SUBAPPLICATION logiBUS_AI_Calibrate_3P_Remote_IDA_OPC (* 3-Punkt-Kalibrierung (AR_CALIBRATE_3P_REF, unabhaengig gespeicherte Rohwerte X_MIN/X_MID/X_MAX + Referenzwerte MIN_REF/MID_REF/MAX_REF alle INI-persistiert) auf VT-Zahlenfelder (Rohwert + kalibrierter Wert, je eigene CNumberVariable) + Bargraph (kalibriert) + 3 VT-Tasten (C_MIN/C_MID/C_MAX) + OPC-UA (Rohwert DWORD + kalibrierter Wert REAL, generisch, ein Kanal). Wie logiBUS_AI_Calibrate_3P_IDA_OPC, aber der Rohwert kommt per Remote-Subscribe (AD_SUBSCRIBE_1) statt von einem lokalen logiBUS_AI_IDA - fuer Sensoren, deren physischer Analog-Eingang auf einer Station OHNE VT-Anschluss sitzt (z.B. Hangausgleich-Winkelsensor B14 auf APIXON STG3, waehrend Kalibrierung+VT auf der Station mit VT-Anschluss laufen). Der Rohwert wird dort per logiBUS_AI_Raw_Publish_OPC publiziert. *)
  (* Standard: 61499-2; Description: Copyright (c) 2026 Meisterschulen am Ostbahnhof This program and the accompanying materials are made available under the terms of the Eclipse Public License 2.0 which is available at https://www.eclipse.org/legal/epl-2.0/ SPDX-License-Identifier: EPL-2.0 *)
  (* Version 1.3, 2026-09-18, Franz Höpfinger, Meisterschulen am Ostbahnhof, AR_CALIBRATE_3P_REF.C_MIN/C_MID/C_MAX von AX-Sockets auf reine EventInputs umgestellt (Franz-Entscheidung, siehe AR_CALIBRATE_2P_REF) - AX_BOOL_TO_X_MIN/_MID/_MAX entfallen ersatzlos, die Merge-Ketten verbinden jetzt direkt per EventConnection mit CALIBRATE.C_MIN/C_MID/C_MAX. *)
  (* Version 1.4, 2026-09-18, Franz Höpfinger, Meisterschulen am Ostbahnhof, C_MIN/C_MAX-Merge-Ketten (2x E_MERGE_2 in Reihe) durch je einen E_MERGE_3 ersetzt, C_MID-Kette (3x E_MERGE_2) durch einen E_MERGE_4 - OR-Merge ist assoziativ, funktional identisch. Siehe logiBUS_AI_Calibrate_IDA_OPC v1.4. *)
  (* Version 1.2, 2026-09-16, Franz Höpfinger, Meisterschulen am Ostbahnhof, Fix (4diac-IDE-Validierungsfehler 'Cannot convert from AR2 to AR'): MID_REF_LIT.VALUEO/MAX_REF_LIT.VALUEO sind bidirektionale AR2-Plugs (Live-VT-Edit + Persistierung), kein einfacher AR-Wert wie CALIBRATE.Y - ein AR_SPLIT_2 direkt dazwischen ist falsch. MIDREF_OUT/MAXREF_OUT werden jetzt stattdessen von den neuen VALUE_OUT-Plugs auf MID_REF_LIT/MAX_REF_LIT gespeist (NumericValue_TO_AR2_OPC Version 1.1, plain-AR-Spiegel des Werts, unabhaengig vom bidirektionalen VALUEO). CAL_OUT (AR_SPLIT_3 auf CALIBRATE.Y, einfacher AR-Wert) war von diesem Fehler nicht betroffen und bleibt unveraendert. *)
  (* Version 1.1, 2026-09-16, Franz Höpfinger, Meisterschulen am Ostbahnhof, Neue optionale Ausgangs-Plugs CAL_OUT/MIDREF_OUT/MAXREF_OUT ergaenzt (AR_SPLIT_2 zu AR_SPLIT_3 fuer CAL, je 1 neuer AR_SPLIT_2 fuer MIDREF/MAXREF dazwischengesetzt) - damit externe Consumer (z.B. Fuellband_Oben_Erkennung/Befuellautomatik fuer den Fuellband-Kanal) den bereits kalibrierten Wert per Adapterverbindung lesen koennen statt selbst nochmal denselben OPC-UA-Knoten lokal zu abonnieren (FORTE: 'Cannot add another one'). Unverdrahtet lassen, wenn nicht gebraucht (z.B. Hangausgleich-Kanal). Siehe BERICHT_2026-09-16_STG3_I1_I3_I4_I6_STALE_REMOTE_SUBSCRIBE.md Abschnitt 16-17 Gruppe C. *)
  (* Version 1.0, 2026-09-11, Franz Höpfinger, Meisterschulen am Ostbahnhof, Remote-Rohwert-Variante von logiBUS_AI_Calibrate_3P_IDA_OPC - logiBUS_AI_IDA+AD_SPLIT_2+AD_PUBLISH_RAW durch AD_SUBSCRIBE_1 ersetzt, Rest der Kalibrier-/VT-Kette unveraendert. Fuer Hangausgleich-Winkelsensor B14 (STG3), Kalibrierung+VT auf STG1. *)
  (* Version 1.6, 2026-09-21, Franz Höpfinger, Meisterschulen am Ostbahnhof, Code-Review-Fund (PR #260): INI_X_MID/INI_X_MAX.DEFAULT_VALUE standen auf REAL#0.5/1.0 statt 0.0 - AR_CALIBRATE_3P_REF's xMidCal/xMaxCal-Kalibriert-Flags latchten dadurch bei JEDEM Boot sofort TRUE, obwohl MID/MAX nie kalibriert wurden. Defaults auf REAL#0.0 korrigiert. Betrifft Hangausgleich. *)
  (* Version 1.5, 2026-09-21, Franz Höpfinger, Meisterschulen am Ostbahnhof, AR_CALIBRATE_3P_REF hat jetzt ein INIT/QI/QO-Enable-Pattern (Bugfix MIN-vor-MID + xClipping) - CALIBRATE bekommt Parameter QI=TRUE, sonst bleibt die FB im START-Zustand haengen und REQ laeuft nie. *)
  PACKAGE MyLib::sys;
  IMPORT isobus::UT::Q::const::IDs::ID_NULL;
  IMPORT logiBUS::utils::conversion::phys::NumericObjectPool_S;
  IMPORT isobus::UT::io::Button::ButtonActivationCode::BT_PRESSED_LATCHED;
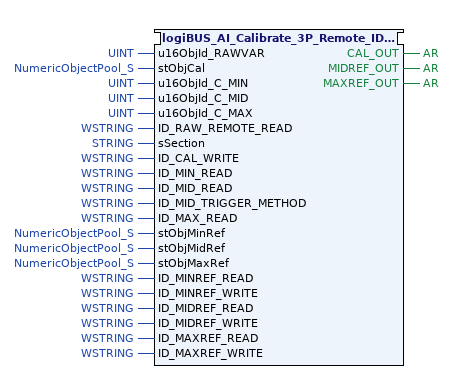
  VAR_INPUT
    u16ObjId_RAWVAR : UINT := ID_NULL; (* Object ID CNumberVariable (Rohwert 0-4095, unkalibriert, reine Diagnose-Anzeige) *)
    stObjCal : logiBUS::utils::conversion::phys::NumericObjectPool_S := (u16ObjId := ID_NULL, r32Scale := 1.0, i32Offset := 0, u8Decimals := 1); (* Object ID + Scale/Offset/Decimals CNumberVariable (kalibrierter Wert, eigene, unabhaengige CNumberVariable) *)
    u16ObjId_C_MIN : UINT := ID_NULL; (* Object ID Taste 'C_MIN' (Min-Position anfahren, dann druecken) *)
    u16ObjId_C_MID : UINT := ID_NULL; (* Object ID Taste 'C_MID' (Mittelstellung anfahren, dann druecken) *)
    u16ObjId_C_MAX : UINT := ID_NULL; (* Object ID Taste 'C_MAX' (Max-Position anfahren, dann druecken) *)
    ID_RAW_REMOTE_READ : WSTRING; (* Remote-Subscribe-Adresse des Rohwerts (DWORD 0-4095, ACTION=SUBSCRIBE) - Gegenstueck zu ID_RAW_WRITE auf der Sensor-Station (logiBUS_AI_Raw_Publish_OPC) *)
    sSection : STRING; (* INI-Sektionsname fuer X_MIN/X_MID/X_MAX/MIN_REF/MID_REF/MAX_REF-Persistenz - pro Kanal eindeutig, sonst kollidieren die Kanaele in settings.ini *)
    ID_CAL_WRITE : WSTRING; (* Kalibrierter-Wert-Ruckmelde-Adresse (REAL, ACTION=PUBLISH) *)
    ID_MIN_READ : WSTRING; (* Remote-C_MIN-Adresse (BOOL, ACTION=SUBSCRIBE, togglet Kalibrier-Min-Trigger wie ein Tastendruck - Web-Client schreibt bei jedem Klick den invertierten letzten Wert, jede Flanke loest C_MIN aus) *)
    ID_MID_READ : WSTRING; (* Remote-C_MID-Adresse (BOOL, ACTION=SUBSCRIBE, siehe ID_MIN_READ) *)
    ID_MID_TRIGGER_METHOD : WSTRING; (* Lokale Methodenadresse (ACTION=CREATE_METHOD) fuer den argument- und rueckgabewertlosen C_MID-Trigger - von einem lokalen CLIENT_0 (z.B. Fahrwerk_Mittelpunkt_Automatik.SUB) per CALL_METHOD aufgerufen, loest wie Button_C_MID/ID_MID_READ ebenfalls C_MID aus *)
    ID_MAX_READ : WSTRING; (* Remote-C_MAX-Adresse (BOOL, ACTION=SUBSCRIBE, siehe ID_MIN_READ) *)
    stObjMinRef : logiBUS::utils::conversion::phys::NumericObjectPool_S := (u16ObjId := ID_NULL, r32Scale := 1.0, i32Offset := 0, u8Decimals := 1); (* Object ID + Scale/Offset/Decimals CNumberVariable (MIN_REF-Referenzwert, VT-Eingabefeld + OPC-UA) *)
    stObjMidRef : logiBUS::utils::conversion::phys::NumericObjectPool_S := (u16ObjId := ID_NULL, r32Scale := 1.0, i32Offset := 0, u8Decimals := 1); (* Object ID + Scale/Offset/Decimals CNumberVariable (MID_REF-Referenzwert, VT-Eingabefeld + OPC-UA) *)
    stObjMaxRef : logiBUS::utils::conversion::phys::NumericObjectPool_S := (u16ObjId := ID_NULL, r32Scale := 1.0, i32Offset := 0, u8Decimals := 1); (* Object ID + Scale/Offset/Decimals CNumberVariable (MAX_REF-Referenzwert, VT-Eingabefeld + OPC-UA) *)
    ID_MINREF_READ : WSTRING; (* Remote-Subscribe-Adresse MIN_REF-Referenzwert (REAL, ACTION=SUBSCRIBE) *)
    ID_MINREF_WRITE : WSTRING; (* Remote-Echo-Adresse MIN_REF-Referenzwert (REAL, ACTION=PUBLISH) *)
    ID_MIDREF_READ : WSTRING; (* Remote-Subscribe-Adresse MID_REF-Referenzwert (REAL, ACTION=SUBSCRIBE) *)
    ID_MIDREF_WRITE : WSTRING; (* Remote-Echo-Adresse MID_REF-Referenzwert (REAL, ACTION=PUBLISH) *)
    ID_MAXREF_READ : WSTRING; (* Remote-Subscribe-Adresse MAX_REF-Referenzwert (REAL, ACTION=SUBSCRIBE) *)
    ID_MAXREF_WRITE : WSTRING; (* Remote-Echo-Adresse MAX_REF-Referenzwert (REAL, ACTION=PUBLISH) *)
  END_VAR
  PLUGS
    CAL_OUT : adapter::types::unidirectional::AR; (* Optional: kalibrierter Wert (= CALIBRATE.Y) fuer externe Consumer, statt eigenem lokalen OPC-UA-Self-Subscribe auf ID_CAL_WRITE. Unverdrahtet lassen, wenn nicht gebraucht. *)
    MIDREF_OUT : adapter::types::unidirectional::AR; (* Optional: live MID_REF-Referenzwert (= MID_REF_LIT.VALUE_OUT, plain-AR-Spiegel des bidirektionalen VALUEO) fuer externe Consumer. Unverdrahtet lassen, wenn nicht gebraucht. *)
    MAXREF_OUT : adapter::types::unidirectional::AR; (* Optional: live MAX_REF-Referenzwert (= MAX_REF_LIT.VALUE_OUT, plain-AR-Spiegel des bidirektionalen VALUEO) fuer externe Consumer. Unverdrahtet lassen, wenn nicht gebraucht. *)
  END_PLUGS
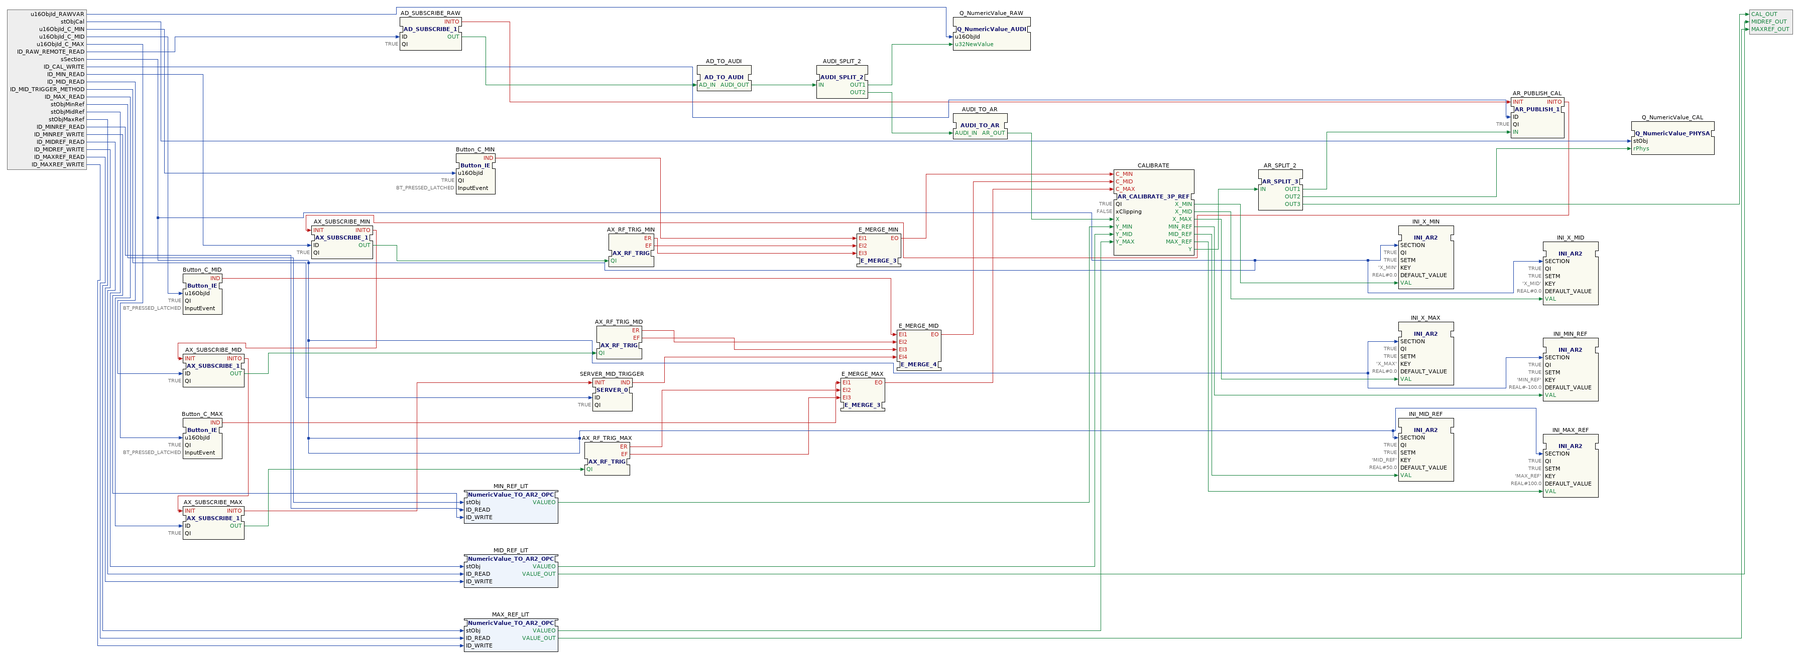
  FBS
    AD_SUBSCRIBE_RAW : adapter::net::AD_SUBSCRIBE_1(QI := TRUE);
    AD_TO_AUDI : adapter::conversion::unidirectional::AD_TO_AUDI;
    AUDI_SPLIT_2 : adapter::events::unidirectional::AUDI_SPLIT_2;
    Q_NumericValue_RAW : isobus::UT::Q::Q_NumericValue_AUDI;
    AUDI_TO_AR : adapter::conversion::unidirectional::AUDI_TO_AR;
    CALIBRATE : adapter::Engineering::measurements::AR_CALIBRATE_3P_REF(QI := TRUE, xClipping := FALSE);
    Button_C_MIN : isobus::UT::io::Button::Button_IE(QI := TRUE, InputEvent := BT_PRESSED_LATCHED);
    Button_C_MID : isobus::UT::io::Button::Button_IE(QI := TRUE, InputEvent := BT_PRESSED_LATCHED);
    Button_C_MAX : isobus::UT::io::Button::Button_IE(QI := TRUE, InputEvent := BT_PRESSED_LATCHED);
    AX_SUBSCRIBE_MIN : adapter::net::AX_SUBSCRIBE_1(QI := TRUE);
    AX_RF_TRIG_MIN : adapter::events::unidirectional::AX_RF_TRIG;
    E_MERGE_MIN : iec61499::events::E_MERGE_3;
    AX_SUBSCRIBE_MID : adapter::net::AX_SUBSCRIBE_1(QI := TRUE);
    AX_RF_TRIG_MID : adapter::events::unidirectional::AX_RF_TRIG;
    SERVER_MID_TRIGGER : iec61499::net::SERVER_0(QI := TRUE);
    E_MERGE_MID : iec61499::events::E_MERGE_4;
    AX_SUBSCRIBE_MAX : adapter::net::AX_SUBSCRIBE_1(QI := TRUE);
    AX_RF_TRIG_MAX : adapter::events::unidirectional::AX_RF_TRIG;
    E_MERGE_MAX : iec61499::events::E_MERGE_3;
    INI_X_MIN : eclipse4diac::storage::INI_AR2(QI := TRUE, SETM := TRUE, KEY := 'X_MIN', DEFAULT_VALUE := REAL#0.0);
    INI_X_MID : eclipse4diac::storage::INI_AR2(QI := TRUE, SETM := TRUE, KEY := 'X_MID', DEFAULT_VALUE := REAL#0.0);
    INI_X_MAX : eclipse4diac::storage::INI_AR2(QI := TRUE, SETM := TRUE, KEY := 'X_MAX', DEFAULT_VALUE := REAL#0.0);
    INI_MIN_REF : eclipse4diac::storage::INI_AR2(QI := TRUE, SETM := TRUE, KEY := 'MIN_REF', DEFAULT_VALUE := REAL#-100.0);
    INI_MID_REF : eclipse4diac::storage::INI_AR2(QI := TRUE, SETM := TRUE, KEY := 'MID_REF', DEFAULT_VALUE := REAL#50.0);
    INI_MAX_REF : eclipse4diac::storage::INI_AR2(QI := TRUE, SETM := TRUE, KEY := 'MAX_REF', DEFAULT_VALUE := REAL#100.0);
    AR_SPLIT_2 : adapter::events::unidirectional::AR_SPLIT_3;
    AR_PUBLISH_CAL : adapter::net::AR_PUBLISH_1(QI := TRUE);
    Q_NumericValue_CAL : isobus::UT::Q::Q_NumericValue_PHYSA;
  END_FBS
  SUBAPPS
    MIN_REF_LIT : MyLib::sys::NumericValue_TO_AR2_OPC;
    MID_REF_LIT : MyLib::sys::NumericValue_TO_AR2_OPC;
    MAX_REF_LIT : MyLib::sys::NumericValue_TO_AR2_OPC;
  END_SUBAPPS
  EVENT_CONNECTIONS
    AD_SUBSCRIBE_RAW.INITO TO AR_PUBLISH_CAL.INIT;
    AR_PUBLISH_CAL.INITO TO AX_SUBSCRIBE_MIN.INIT;
    AX_SUBSCRIBE_MIN.INITO TO AX_SUBSCRIBE_MID.INIT;
    AX_SUBSCRIBE_MID.INITO TO AX_SUBSCRIBE_MAX.INIT;
    AX_SUBSCRIBE_MAX.INITO TO SERVER_MID_TRIGGER.INIT;
    Button_C_MIN.IND TO E_MERGE_MIN.EI1;
    AX_RF_TRIG_MIN.ER TO E_MERGE_MIN.EI2;
    AX_RF_TRIG_MIN.EF TO E_MERGE_MIN.EI3;
    E_MERGE_MIN.EO TO CALIBRATE.C_MIN;
    Button_C_MID.IND TO E_MERGE_MID.EI1;
    AX_RF_TRIG_MID.ER TO E_MERGE_MID.EI2;
    AX_RF_TRIG_MID.EF TO E_MERGE_MID.EI3;
    SERVER_MID_TRIGGER.IND TO E_MERGE_MID.EI4;
    E_MERGE_MID.EO TO CALIBRATE.C_MID;
    Button_C_MAX.IND TO E_MERGE_MAX.EI1;
    AX_RF_TRIG_MAX.ER TO E_MERGE_MAX.EI2;
    AX_RF_TRIG_MAX.EF TO E_MERGE_MAX.EI3;
    E_MERGE_MAX.EO TO CALIBRATE.C_MAX;
  END_CONNECTIONS
  DATA_CONNECTIONS
    u16ObjId_RAWVAR TO Q_NumericValue_RAW.u16ObjId;
    stObjCal TO Q_NumericValue_CAL.stObj;
    u16ObjId_C_MIN TO Button_C_MIN.u16ObjId;
    u16ObjId_C_MID TO Button_C_MID.u16ObjId;
    u16ObjId_C_MAX TO Button_C_MAX.u16ObjId;
    ID_RAW_REMOTE_READ TO AD_SUBSCRIBE_RAW.ID;
    sSection TO INI_X_MIN.SECTION;
    sSection TO INI_X_MID.SECTION;
    sSection TO INI_X_MAX.SECTION;
    sSection TO INI_MIN_REF.SECTION;
    sSection TO INI_MID_REF.SECTION;
    sSection TO INI_MAX_REF.SECTION;
    ID_CAL_WRITE TO AR_PUBLISH_CAL.ID;
    ID_MIN_READ TO AX_SUBSCRIBE_MIN.ID;
    ID_MID_READ TO AX_SUBSCRIBE_MID.ID;
    ID_MID_TRIGGER_METHOD TO SERVER_MID_TRIGGER.ID;
    ID_MAX_READ TO AX_SUBSCRIBE_MAX.ID;
    stObjMinRef TO MIN_REF_LIT.stObj;
    ID_MINREF_READ TO MIN_REF_LIT.ID_READ;
    ID_MINREF_WRITE TO MIN_REF_LIT.ID_WRITE;
    stObjMidRef TO MID_REF_LIT.stObj;
    ID_MIDREF_READ TO MID_REF_LIT.ID_READ;
    ID_MIDREF_WRITE TO MID_REF_LIT.ID_WRITE;
    stObjMaxRef TO MAX_REF_LIT.stObj;
    ID_MAXREF_READ TO MAX_REF_LIT.ID_READ;
    ID_MAXREF_WRITE TO MAX_REF_LIT.ID_WRITE;
  END_CONNECTIONS
  ADAPTER_CONNECTIONS
    AD_SUBSCRIBE_RAW.OUT TO AD_TO_AUDI.AD_IN;
    AD_TO_AUDI.AUDI_OUT TO AUDI_SPLIT_2.IN;
    AUDI_SPLIT_2.OUT1 TO Q_NumericValue_RAW.u32NewValue;
    AUDI_SPLIT_2.OUT2 TO AUDI_TO_AR.AUDI_IN;
    AUDI_TO_AR.AR_OUT TO CALIBRATE.X;
    CALIBRATE.X_MIN TO INI_X_MIN.VAL;
    CALIBRATE.X_MID TO INI_X_MID.VAL;
    CALIBRATE.X_MAX TO INI_X_MAX.VAL;
    CALIBRATE.MIN_REF TO INI_MIN_REF.VAL;
    CALIBRATE.MID_REF TO INI_MID_REF.VAL;
    CALIBRATE.MAX_REF TO INI_MAX_REF.VAL;
    MIN_REF_LIT.VALUEO TO CALIBRATE.Y_MIN;
    MID_REF_LIT.VALUEO TO CALIBRATE.Y_MID;
    MID_REF_LIT.VALUE_OUT TO MIDREF_OUT;
    MAX_REF_LIT.VALUEO TO CALIBRATE.Y_MAX;
    MAX_REF_LIT.VALUE_OUT TO MAXREF_OUT;
    CALIBRATE.Y TO AR_SPLIT_2.IN;
    AR_SPLIT_2.OUT1 TO AR_PUBLISH_CAL.IN;
    AR_SPLIT_2.OUT2 TO Q_NumericValue_CAL.rPhys;
    AR_SPLIT_2.OUT3 TO CAL_OUT;
    AX_SUBSCRIBE_MIN.OUT TO AX_RF_TRIG_MIN.QI;
    AX_SUBSCRIBE_MID.OUT TO AX_RF_TRIG_MID.QI;
    AX_SUBSCRIBE_MAX.OUT TO AX_RF_TRIG_MAX.QI;
  END_CONNECTIONS
END_SUBAPPLICATION
